INTERFACE I_SessionManager

METHOD PUBLIC CreateSession : T_MAXSTRING
END_METHOD

METHOD PUBLIC DisposeAllSessions
VAR_INPUT
END_VAR
END_METHOD

METHOD PUBLIC IsValidSession : BOOL
VAR_INPUT
	Id : T_MAXSTRING;
END_VAR
END_METHOD

METHOD PUBLIC RefreshSession
VAR_INPUT
	Id : T_MAXSTRING;
END_VAR
END_METHOD

END_INTERFACE

(* stored: Version 1.1.0.1, ProductVersion 3.1.4026.13
   Itf I_SessionManager: Id {17facafb-fc5c-45f8-9123-2272195bc402}
   Method CreateSession: Id {bd9d747e-a1a8-40c9-a57f-2d82c9c2e236}
   Method DisposeAllSessions: Id {540dc239-d8a3-4404-8c22-d1497f8096c7}
   Method IsValidSession: Id {9e2cb71c-e925-4328-bdbe-dadf6a82fb19}
   Method RefreshSession: Id {7e866d52-51ae-49fd-9464-41824a5733ef} *)
